FUNCTION_BLOCK Factory
VAR
	ObjPtr : POINTER TO BasicObject;
END_VAR

METHOD Create : ITF_Cyclic
VAR_INPUT
END_VAR
ObjPtr := __NEW(BasicObject);
Create := ObjPtr^;
END_METHOD

END_FUNCTION_BLOCK

(* stored: Version 1.1.0.1, ProductVersion 3.1.4024.12
   POU Factory: Id {ce0d4dba-2a11-4e3f-b0cc-8cd3d42ab19b}, SpecialFunc None
   Method Create: Id {849a93e0-0589-496e-8750-c8238abd2149} *)
